TYPE ST_CFG_TurnTable :

STRUCT
	TurnTimeoutValue 			: TIME := T#30S; 			// Timeout value for turning
	TurnBrakeDelayTime			: TIME := T#2S; 			// Turning Brake release time	
	TurnHomePosFree				: E_Positions_TurnControl; // Homeposition turn table when zone free
	TurnHomePosOccupied			: E_Positions_TurnControl; // Homeposition turn table when zone occupied		
END_STRUCT
END_TYPE

(* stored: Version 1.1.0.1, ProductVersion 3.1.4024.9
   DUT ST_CFG_TurnTable: Id {7d394edb-e25a-4f3a-a012-17c70df7b839} *)
